INTERFACE ITF_SwitchStation EXTENDS __SYSTEM.IQueryInterface

METHOD SwitchMoveComplete : BOOL
VAR_INPUT
END_VAR
END_METHOD

END_INTERFACE

(* stored: Version 1.1.0.1, ProductVersion 3.1.4024.11
   Itf ITF_SwitchStation: Id {a4cd9fdb-f0b5-4075-bf63-91413cfe4e9a}
   Method SwitchMoveComplete: Id {3217cd50-c1a2-47a5-b916-b18302ef9cee} *)
